FUNCTION_BLOCK ControlDispenserIncomplete (* Basic Function Block Type *)
  (* Standard: 61499-2 *)
  (* Version 0.3, 2009-09-15, JHC, Holobloc Inc, Changed transition priorities. *)
  (* Version 0.2, 2003-12-04, JHC, Rockwell Automation, Renamed for better indexing. *)
  (* Version 0.1, 2002-11-05, JHC, Rockwell Automation, Corrected missing ST element in Algorithm REQ. *)
  (* Version 0.0, 2000-05-30, JHC, Rockwell Automation *)
  (* Compiler header: package fb.rt.template; *)
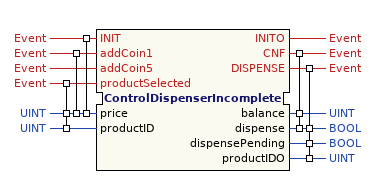
  EVENT_INPUT
    INIT WITH price; (* Initialization Request *)
    addCoin1 WITH price; (* Normal Execution Request *)
    addCoin5;
    productSelected WITH price, productID;
  END_EVENT
  EVENT_OUTPUT
    INITO; (* Initialization Confirm *)
    CNF WITH balance, dispense; (* Execution Confirmation *)
    DISPENSE WITH productIDO, dispense, dispensePending;
  END_EVENT
  VAR_INPUT
    price : UINT; (* Input event qualifier *)
    productID : UINT;
  END_VAR
  VAR_OUTPUT
    balance : UINT;
    dispense : BOOL;
    dispensePending : BOOL;
    productIDO : UINT;
  END_VAR
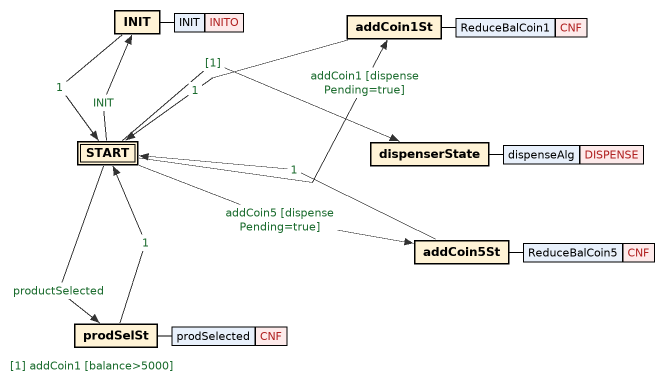
  EC_STATES
    START; (* Initial State *)
    INIT : INIT -> INITO; (* Initialization *)
    prodSelSt : prodSelected -> CNF;
    addCoin1St : ReduceBalCoin1 -> CNF;
    addCoin5St : ReduceBalCoin5 -> CNF;
    dispenserState : dispenseAlg -> DISPENSE;
  END_STATES
  EC_TRANSITIONS
    INIT TO START := 1;
    START TO INIT := INIT;
    START TO prodSelSt := productSelected;
    prodSelSt TO START := 1;
    START TO addCoin1St := addCoin1 [dispensePending=true];
    START TO addCoin5St := addCoin5 [dispensePending=true];
    addCoin5St TO START := 1;
    START TO dispenserState := addCoin1 [balance>5000];
    addCoin1St TO START := 1;
  END_TRANSITIONS
  ALGORITHM INIT IN ST: (* Initialization algorithm *)
balance:=0;
dispensePending:=false;
  END_ALGORITHM
  ALGORITHM ReduceBalCoin1 IN ST:
balance:=balance-1;

IF (balance<=0) THEN
dispense:=true;
END_IF;
  END_ALGORITHM
  ALGORITHM ReduceBalCoin5 IN ST:
balance:=balance-5;
IF (balance<=0) THEN
dispense:=true;
END_IF;
  END_ALGORITHM
  ALGORITHM prodSelected IN ST:
balance:=price;
dispensePending:=true;
productIDO:=productID;
  END_ALGORITHM
  ALGORITHM dispenseAlg IN ST:
dispense:=TRUE;
  END_ALGORITHM
END_FUNCTION_BLOCK
